// TwinCAT 3 PLC project Controller
// ProgramVersion: 3.1.4020.2
// libraries:
//   Tc2_Standard, * (Beckhoff Automation GmbH)
//   Tc2_System, * (Beckhoff Automation GmbH)
//   Tc2_TcpIp, * (Beckhoff Automation GmbH)
//   Tc2_Utilities, * (Beckhoff Automation GmbH)
//   Tc3_Module, * (Beckhoff Automation GmbH)
// project tree:
//   / GlobalTextList.TcGTLO, ImagePool.TcIPO (not stored), PlcTask.TcTTO, Visualization Manager.TcVMO (not stored), VISU_TASK.TcTTO
//   GVLs/ GVL.TcGVL
//   POUs/Helpers/ FB_FrameFifo.TcPOU, FB_LogFifo.TcPOU
//   POUs/ MAIN.TcPOU
//   POUs/SocketClient/ FB_ProcessSocketData.TcPOU, FB_SocketClient.TcPOU, FB_SocketClientConnection.TcPOU
//   VISUs/ Visualization.TcVIS
// real-time tasks:
//   TASK PlcTask: cycle T#10ms, priority 20, ADS port 350
//   TASK IOTask: cycle T#10ms, priority 1, ADS port 351
//   TASK VISU_TASK: cycle T#200000us, priority 30, ADS port 352

CONFIGURATION Controller
    RESOURCE PLC ON TwinCAT3
        TASK PlcTask(INTERVAL := T#10ms, PRIORITY := 20);
        TASK VISU_TASK(INTERVAL := T#200000us, PRIORITY := 30);
        PROGRAM MAIN WITH PlcTask : MAIN;
        PROGRAM VisuElems_Visu_Prg WITH VISU_TASK : VisuElems.Visu_Prg;
    END_RESOURCE
END_CONFIGURATION

// ---- GVLs/GVL.TcGVL
{attribute 'qualified_only'}
VAR_GLOBAL CONSTANT
	PLCPRJ_BUFFER_SIZE		: UDINT := 1000;					(* Max. internal fifo/receiver buffer size *)
	
	PLCPRJ_CLIENT_SEND_CYCLE_TIME			: TIME := T#1S;
	PLCPRJ_RECEIVE_POLLING_TIME				: TIME := T#100MS;
	PLCPRJ_RECEIVE_TIMEOUT					: TIME := T#50S;
	
	(* Some project specific error codes *)
	PLCPRJ_ERROR_RECEIVE_TIMEOUT			: UDINT := 16#8101;(* Receive timeout *)
	PLCPRJ_ERROR_SENDFIFO_OVERFLOW			: UDINT := 16#8102;(* Send fifo overflow *)
	PLCPRJ_ERROR_RECFIFO_OVERFLOW			: UDINT := 16#8103;(* Receive fifo overflow *)	
	
	TERMINATION_CHAR_CODE					: BYTE := 10;	
	
END_VAR

VAR_GLOBAL
	sSrvNetID					: T_AmsNetID	:= ''; 				(* TwinCAT TCP/IP server network address - Set to Local via ''*)
	sSocketRemoteHost			: T_IPv4Addr := '10.5.1.166';		(* Remote Socket Server IP Address*)
	nSocketRemotePort			: UDINT := 14150;  					(* Server port number *)
	
	RFID_TAG			AT %Q*	: STRING(40);
	READ_ZONE_BEGIN 	AT %I*	: BOOL;
	SET_TEST_OUTPUT		AT %Q* 	: BOOL;
	TON_FLASH					: TON;
	
END_VAR

// ---- POUs/MAIN.TcPOU
PROGRAM MAIN
VAR
	bSocketCloseAll			: BOOL := TRUE;
	fbSocketCloseAll		: FB_SocketCloseAll;
	fbSocketClient			: FB_SocketClient := ( 	sRemoteHost := GVL.sSocketRemoteHost,(* Remote (server) IP address! *)
										nRemotePort := GVL.nSocketRemotePort,(* Remote (server) port number! *)  
										sPrefix := 'CLIENT::' );(* Application (connection) instance *)
										
	bEnableSocket			: BOOL 	:= TRUE;   (* TRUE => enable client data exchange, FALSE => disable *)
	bEnableLogging			: BOOL	:= TRUE;   (* TRUE => Enable message/error log, FALSE => Disable *)
END_VAR

(* On PLC reset or program download close all old (opened) connections *)
fbSocketCloseAll( 	sSrvNetID := GVL.sSrvNetID, 
					bExecute:= bSocketCloseAll );
					
IF fbSocketCloseAll.bBusy OR fbSocketCloseAll.bError THEN
	RETURN;
END_IF
bSocketCloseAll := FALSE;

fbSocketClient( sSrvNetId := GVL.sSrvNetID, 
				bEnable := bEnableSocket, 
				bLog := bEnableLogging );
				
IF GVL.TON_FLASH.Q THEN
	GVL.TON_FLASH( IN := FALSE);
	GVL.SET_TEST_OUTPUT := 0;
END_IF

END_PROGRAM

// ---- POUs/SocketClient/FB_SocketClient.TcPOU
FUNCTION_BLOCK FB_SocketClient
VAR_INPUT
	sSrvNetID	: T_AmsNetID	:= '';(* TwinCAT TCP/IP server network address *)
	sRemoteHost	: T_IPv4Addr 	:= '127.0.0.1';(* Server network address *)
	nRemotePort	: UDINT 		:= 200;(* Server port number *)
	bEnable		: BOOL 			:= FALSE;(* TRUE => enable client data exchange, FALSE => disable *)
	bLog		: BOOL 			:= FALSE;(* TRUE => Enable log message output, FALSE => Disable *)
	sPrefix		: STRING 		:= 'CLIENT::';(* Log message description string (allows the identification of log message source) *)
END_VAR
VAR_OUTPUT
	eState		: E_SocketConnectionState := eSOCKET_DISCONNECTED;(* TCP/IP connection state *)
END_VAR
VAR
	fbProcessSocketData : FB_ProcessSocketData;				(* Client application control function block *)
	fbClientConnection	: FB_SocketClientConnection;		(* Client data exchange control function block *)
	fbTx 				: FB_FrameFifo;						(* Tx fifo *)
	fbRx 				: FB_FrameFifo;						(* Rx fifo *)
	fbLog				: FB_LogFifo;						(* Log/debug/error fifo *)
END_VAR

(*-------------------------- Trigger data exchange -----------------------------------------------*)
fbClientConnection( sSrvNetID := sSrvNetID, fbRx := fbRx, fbTx := fbTx, fbLog := fbLog, 
					bEnable := bEnable, sRemoteHost := sRemoteHost, nRemotePort := nRemotePort,  
					bLog := bLog, sPrefix := sPrefix, eState=>eState );
	
IF fbClientConnection.eState = eSOCKET_CONNECTED THEN (* Connection established *)
	fbProcessSocketData( fbTx := fbTx, fbRx := fbRx, fbLog := fbLog );
END_IF

END_FUNCTION_BLOCK

// ---- POUs/SocketClient/FB_ProcessSocketData.TcPOU
FUNCTION_BLOCK FB_ProcessSocketData
VAR_IN_OUT
	fbTx 		: FB_FrameFifo;(* TX fifo *)
	fbRx 		: FB_FrameFifo;(* RX fifo *)
	fbLog		: FB_LogFifo;(* Log message fifo *)
END_VAR
VAR
	sToServer	: T_MaxString := '';
	sFromServer	: T_MaxString := '';
	sLogMessage : T_MaxString := '';
	nCounter	: UDINT;
	fbSndTimer	: TON;
END_VAR

(*------------------------------- Send cyclic message strings ------------------------------------------*)
fbSndTimer( IN := FALSE, PT := GVL.PLCPRJ_CLIENT_SEND_CYCLE_TIME );
IF fbSndTimer.Q THEN
	fbSndTimer( IN := FALSE );

	(* Create new message string *)
	nCounter := nCounter  + 1;
	sToServer := CONCAT( 'Client message: ', UDINT_TO_STRING(nCounter) );

	fbTx.AddToTail( sPut := sToServer );(* Put string to the tx fifo *)
	IF NOT fbTx.bOk THEN(* TX fifo overflow => log error *)
		fbLog.Error( sMessage := 'FB_FrameFifo(sender)', nErrID := GVL.PLCPRJ_ERROR_SENDFIFO_OVERFLOW );
	END_IF

END_IF

(*------------------------------- Get received message strings ------------------------------------------*)
REPEAT
	fbRx.RemoveFromHead();(* Fetch string from rx fifo *)
	IF fbRx.bOk THEN(* Success *)

		(* TODO: Implement receive data handler *)
		sFromServer := fbRx.sGet;
		
		(* TEST HANDLER *)
		GVL.RFID_TAG := sFromServer;
		IF LEN(sFromServer) > 0 THEN
			GVL.TON_FLASH( IN := TRUE, PT := T#0.25S );		
			GVL.SET_TEST_OUTPUT := 1;	
		END_IF
		sFromServer := '';
		(* END TEST HANDLER *)
		
	END_IF
	
UNTIL NOT fbRx.bOk

END_REPEAT


(*------------------------------- Get log/error messages from log fifo ------------------------------------------*)
REPEAT
	fbLog.Remove( );
	IF fbLog.bOk THEN

		(* TODO: Implement log message handler *)
		sLogMessage := fbLog.sGet;

	END_IF
UNTIL NOT fbLog.bOk
END_REPEAT

END_FUNCTION_BLOCK

// ---- POUs/Helpers/FB_FrameFifo.TcPOU
(* Tx/Rx (string data) fifo control function block *)
FUNCTION_BLOCK FB_FrameFifo
VAR_INPUT
	bLog		: BOOL			:= FALSE;			(* TRUE => Enable log message output, FALSE => Disable *)
	sPrefix		: STRING		:= 'Unknown::';		(* Log message description string (allows the identification of log message source) *)
	sPut		: T_MaxString 	:= ''; 				(* String message to add (write) to the fifo *)
END_VAR
VAR_OUTPUT
	bOk			: BOOL; 	 						(* TRUE = New entry added or removed succesfully, FALSE = Fifo overflow or fifo empty *)
	sGet		: T_MaxString 	:= '';				(* String message removed (read) from fifo *)
	nCount		: UDINT			:= 0;				(* Number of fifo entries *)
	cbFree		: UDINT 		:= 0;				(* Free buffer space *)	
END_VAR
VAR
	fbBuffer 	: FB_StringRingBuffer := (bOverwrite := FALSE);(* Basic (lower level) string buffer control function block *)
	buffer		: ARRAY[-3..GVL.PLCPRJ_BUFFER_SIZE] OF BYTE;(* Internal buffer memory *)	
END_VAR

;

ACTION AddToTail:
(* Adds new fifo entry *)
fbBuffer.A_AddTail( pBuffer:= ADR(buffer), cbBuffer:= SIZEOF(buffer),
					putValue:= sPut, bOk=>bOk, nCount=>nCount );
IF bOk THEN
	cbFree := GVL.PLCPRJ_BUFFER_SIZE - fbBuffer.cbSize;(* Calculate the free buffer space *)
	IF bLog THEN(* Log message *)
		ADSLOGSTR( ADSLOG_MSGTYPE_HINT OR ADSLOG_MSGTYPE_LOG, CONCAT( sPrefix, '<="%s"' ), sPut );
	END_IF
END_IF
END_ACTION

ACTION Clear:
(* Resets fifo = clears all data *)
fbBuffer.A_Reset( pBuffer:= ADR(buffer), cbBuffer:= SIZEOF(buffer),
				bOk=>bOk, getValue=>sGet, nCount=>nCount );
				
cbFree := GVL.PLCPRJ_BUFFER_SIZE;(* Free buffer size *)
END_ACTION

ACTION RemoveFromHead:
(* Removes oldest fifo entry *)
fbBuffer.A_RemoveHead( pBuffer:= ADR(buffer), cbBuffer:= SIZEOF(buffer),
						bOk=>bOk, getValue=>sGet, nCount=>nCount );
IF bOk THEN
	cbFree := GVL.PLCPRJ_BUFFER_SIZE - fbBuffer.cbSize;(* Calculate the free buffer space *)
END_IF
END_ACTION

END_FUNCTION_BLOCK

// ---- POUs/Helpers/FB_LogFifo.TcPOU
(* Log/debug/error message fifo *)
FUNCTION_BLOCK FB_LogFifo
VAR_INPUT
	bLog		: BOOL 		:= FALSE;				(* TRUE => Enable log message output, FALSE => Disable *)
	sPrefix		: STRING 	:= 'Unknown::';			(* Log message description string (allows the identification of log message source) *)
	
	sMessage	: STRING 	:= '';					(* String message to add (write) to the fifo *)
	nErrID		: UDINT 	:= 0;					(* Error code to add (write) to the fifo *)
	hSocket		: T_HSOCKET;						(* Socket connection handle *)
END_VAR
VAR_OUTPUT
	bOk			: BOOL;								(* TRUE = New entry added or removed succesfully, FALSE = Fifo overflow or fifo empty *)
	sGet		: T_MaxString := '';				(* String entry removed (read) from fifo *)
	nCount		: UDINT := 0;						(* Number of fifo entries *)	
END_VAR
VAR
	fbBuffer 	: FB_StringRingBuffer;(* Basic (lower level) string buffer control function block *)
	buffer		: ARRAY[0..GVL.PLCPRJ_BUFFER_SIZE] OF BYTE;(* Internal buffer memory *)
	sSource		: T_MaxString;	
	sPut		: T_MaxString;	
END_VAR

;

ACTION Clear:
(* Clears all fifo entries *)
fbBuffer.A_Reset( 	pBuffer := ADR( buffer ), cbBuffer := SIZEOF( buffer ), 
					bOk=>bOk, nCount=>nCount, getValue=>sGet );
END_ACTION

ACTION Error:
(* Adds new fifo entry *)
IF nErrID = 0 THEN
	sSource := '::Error: 0x';
ELSIF ( nErrID AND 16#80000000) = 16#80000000 THEN
	IF nErrID = 16#80072746 THEN
		sSource := '::Win32 error (the connection is reset by remote side): 0x';
	ELSE
		sSource := '::Win32 error: 0x';
	END_IF
ELSIF (nErrID AND 16#00008100) = 16#00008100 THEN
	CASE nErrID OF
		GVL.PLCPRJ_ERROR_RECEIVE_TIMEOUT:
			sSource := '::PLC sample project receive timeout error: 0x';
		GVL.PLCPRJ_ERROR_SENDFIFO_OVERFLOW:
			sSource := '::PLC sample project send fifo overflow error: 0x';
		GVL.PLCPRJ_ERROR_RECFIFO_OVERFLOW:
			sSource := '::PLC sample project receive fifo overflow error: 0x';
	ELSE
		sSource := '::Other PLC sample project error: 0x';
	END_CASE
ELSIF (nErrID AND 16#00008000) = 16#00008000 THEN
	sSource := '::Internal TCP/IP Connection Server error: 0x';
ELSE
	sSource := '::TwinCAT System error: 0x';
END_IF

sPut := CONCAT( CONCAT( CONCAT( sPrefix, sMessage ), sSource ), DWORD_TO_HEXSTR( nErrID AND 16#FFFF, 0, FALSE ) ); 

fbBuffer.A_AddTail( pBuffer:= ADR(buffer), cbBuffer:= SIZEOF(buffer),
					putValue:= sPut, bOk=>bOk, nCount=>nCount );
IF bOk THEN
	IF bLog THEN(* Log error message *)
		ADSLOGSTR( ADSLOG_MSGTYPE_ERROR OR ADSLOG_MSGTYPE_LOG, '%s', sPut );	
	END_IF
END_IF
END_ACTION

ACTION Message:
(* Adds new fifo entry *)
sPut := CONCAT( CONCAT( sPrefix, sMessage ), CONCAT( '::', HSOCKET_TO_STRING(hSocket) ) );
fbBuffer.A_AddTail( pBuffer:= ADR(buffer), cbBuffer:= SIZEOF(buffer),
					putValue:= sPut, bOk=>bOk, nCount=>nCount );
IF bOk THEN
	IF bLog THEN(* Log information message *)
		ADSLOGSTR( ADSLOG_MSGTYPE_HINT OR ADSLOG_MSGTYPE_LOG, '%s', sPut );	
	END_IF
END_IF
END_ACTION

ACTION Remove:
(* Removes oldest fifo entry *)
IF nCount = 0 THEN
	sGet := '';
	bOk := FALSE;
	RETURN;
END_IF

fbBuffer.A_RemoveHead( pBuffer:= ADR(buffer), cbBuffer:= SIZEOF(buffer),
						getValue=>sGet, bOk=>bOk, nCount=>nCount );
END_ACTION

END_FUNCTION_BLOCK

// ---- POUs/SocketClient/FB_SocketClientConnection.TcPOU
(* This function block implements simple TCP/IP client protocol. *)
FUNCTION_BLOCK FB_SocketClientConnection
VAR_IN_OUT
	fbTx 		: FB_FrameFifo;  (* TX fifo *)
	fbRx 		: FB_FrameFifo;  (* RX fifo *)
	fbLog		: FB_LogFifo;    (* Log message fifo *)
END_VAR

VAR_INPUT
	sSrvNetID	: T_AmsNetID	:= '';				(* TwinCAT TCP/IP server network address *)
	sRemoteHost	: T_IPv4Addr	:= '127.0.0.1';		(* Server network address *)
	nRemotePort	: UDINT			:= 200;				(* Remote server port *)
	bEnable		: BOOL			:= FALSE;			(* TRUE => Enable/connect, FALSE => Disable/disconnect *)
	tReconnect	: TIME 			:= T#10S;			(* Try to reconnect after this time *)
	bLog		: BOOL 			:= FALSE;			(* TRUE => Enable log message output, FALSE => Disable *)
	sPrefix		: STRING 		:= 'CLIENT::';		(* Log message description string (allows the identification of log message source) *)
END_VAR

VAR_OUTPUT
	eState		: E_SocketConnectionState := eSOCKET_DISCONNECTED;		(* TCP/IP connection state *)
END_VAR
VAR
	fbSocketConnect 	: FB_ClientServerConnection;					(* Create/release TCP/IP connection *)
	fbSocketSend		: FB_SocketSend;								(* Send TCP/IP data *)
	fbSocketReceive		: FB_SocketReceive;								(* Receive TCP/IP data *)
	
	nState 		: BYTE;													(* Global state *)
	bSndBusy 	: BOOL;													(* Tx state *)
	bRcvBusy 	: BOOL;													(* Rx state *)
	bDisconnect	: BOOL;													(* Disconnect flag, if set the socket will be closed *)

	fbReceivePollTimer	: TON;											(* Receive poll timer *)
	fbResponseTimer		: TON;											(* Response timeout timer *)
	fbReconnectTimer 	: TON;											(* Reconnect timer *)

	dBytesReceived		: UDINT;										(* Count of received data bytes *)
	dRxLength			: UDINT;										(* Byte length of received string *)
	buffer				: ARRAY[0..GVL.PLCPRJ_BUFFER_SIZE] OF BYTE;		(* Temp. RX buffer *)
	sRxFrame			: T_MaxString;
	sTxFrame			: T_MaxString;
	i					: UDINT;
	bAbort				: BOOL;
END_VAR

CASE nState OF
	0:(* Connect *)
		fbSocketConnect( sSrvNetID 		:= sSrvNetID,
						nMode			:= SEL( bLog, 0, CONNECT_MODE_ENABLEDBG),(* Enable/disable debug messages? *)
						sRemoteHost 	:= sRemoteHost, nRemotePort := nRemotePort,
						bEnable			:= bEnable, tReconnect	:= tReconnect,
						eState			=> eState );
						
		IF NOT fbSocketConnect.bBusy THEN
			IF NOT fbSocketConnect.bError THEN
				IF eState = eSOCKET_CONNECTED THEN   (* We are connected *)
					
					fbTx.Clear( sPrefix := CONCAT( sPrefix, 'FB_FrameFifo(sender)::' ), bLog := bLog );(* Clear TX fifo (optional) *)
					fbRx.Clear( sPrefix := CONCAT( sPrefix, 'FB_FrameFifo(receiver)::' ), bLog := bLog );(* Clear RX fifo (optional) *)
					fbLog.Clear( sPrefix := sPrefix, bLog := bLog );(* Clear log fifo (optional) *)
					bSndBusy := FALSE;
					bRcvBusy := FALSE;
					bDisconnect := FALSE;
					dBytesReceived 	:= 0;

					fbReceivePollTimer( IN := FALSE, PT := T#0S );
					fbResponseTimer( IN := FALSE, PT := GVL.PLCPRJ_RECEIVE_TIMEOUT );
					fbReconnectTimer( IN := FALSE, PT := tReconnect );
				
					fbLog.Message( sMessage := 'Connection established!', hSocket := fbSocketConnect.hSocket );
					nState := 1;
				END_IF
			ELSE(* Connect error => log error *)
				fbLog.Error( sMessage := 'FB_ClientServerConnection()', nErrID := fbSocketConnect.nErrId );
			END_IF
		END_IF


	1:(* Data exchange state *)
		bDisconnect := NOT bEnable OR bDisconnect;(* User/internal disconnect requested? *)
		IF bDisconnect AND NOT bSndBusy AND NOT bRcvBusy THEN
			bDisconnect := FALSE;
			fbLog.Message( sMessage := 'Closing connection!', hSocket := fbSocketConnect.hSocket );
			nState := 2;(* Disconnect *)
		ELSE

			(* ------------------ Send tx data -------------------------------------- *)
			
			IF NOT bDisconnect AND NOT bSndBusy THEN
				fbTx.RemoveFromHead( sGet => sTxFrame );(* Remove oldest string entry *)
				IF fbTx.bOk THEN(* Success *)
					fbSocketSend( bExecute := FALSE );
					fbSocketSend(sSrvNetID 	:= sSrvNetID,
							hSocket		:= fbSocketConnect.hSocket,
							cbLen		:= INT_TO_UDINT(LEN( sTxFrame )) + 1,(* Send string inclusive string (null) delimiter! *)
							pSrc		:= ADR( sTxFrame ),(* Address of the string variable *)
							bExecute	:= TRUE );
					bSndBusy := TRUE;
				END_IF
			ELSE(* Wait until send not busy *)
				fbSocketSend( bExecute := FALSE );
				IF NOT fbSocketSend.bBusy THEN
					bSndBusy := FALSE;
					IF fbSocketSend.bError THEN(* Send error => log error and disconnect *)
						fbLog.Error( sMessage := 'FB_SocketSend()', nErrID := fbSocketSend.nErrId );
						bDisconnect := TRUE;(* Set flag *)
					END_IF
				END_IF
			END_IF  
			(* ---------------------------------------------------------------------- *)


			(* ---------------------- Get rx data ----------------------------------- *)
			IF NOT bDisconnect AND NOT bRcvBusy THEN
				
				fbReceivePollTimer( IN := TRUE );
				IF fbReceivePollTimer.Q THEN
					IF fbRx.cbFree >= SIZEOF(sRxFrame) THEN(* Check free rx fifo space *)
						fbReceivePollTimer( IN := FALSE, PT := GVL.PLCPRJ_RECEIVE_POLLING_TIME );
						fbSocketReceive( bExecute := FALSE );
						fbSocketReceive(sSrvNetId	:= sSrvNetID,
										hSocket		:= fbSocketConnect.hSocket,
										cbLen		:= SIZEOF(buffer) - dBytesReceived,
										pDest		:= ADR(buffer) + dBytesReceived,
										bExecute	:= TRUE );
						bRcvBusy := TRUE;
					END_IF
				END_IF
				
			ELSE(* Wait until receive not busy *)

				fbSocketReceive( bExecute := FALSE );
				IF NOT fbSocketReceive.bBusy THEN
					bRcvBusy := FALSE;
					IF NOT fbSocketReceive.bError THEN
						IF fbSocketReceive.nRecBytes > 0 THEN(* Bytes received *)
							
							fbReceivePollTimer( IN := FALSE, PT := T#0S );(* Bytes received => increase the read (polling) speed *)
							fbResponseTimer( IN := FALSE );(* Bytes received => disable timeout check *)
							dBytesReceived := dBytesReceived + fbSocketReceive.nRecBytes;(* Calculate the number of received data bytes *)

							(* Parse received bytes and extract strings *)
							REPEAT
								bAbort := TRUE;(* set flag *)
								IF dBytesReceived > 0 THEN

									(* Search for string null delimiter *)
									FOR i:= 0 TO dBytesReceived - 1 BY 1 DO
										IF buffer[i] = GVL.TERMINATION_CHAR_CODE THEN (* End of string position found *)

											dRxLength := i + 1;(* Calculate the length of string (inclusive the end delimiter) *)
											MEMCPY( ADR(sRxFrame), ADR(buffer), MIN(dRxLength, SIZEOF(sRxFrame) ) );(* Copy string bytes to temp string variable *)

											fbRx.AddToTail( sPut := sRxFrame );(* Add string to the rx fifo *)
											IF fbRx.bOk THEN
												MEMMOVE( ADR(buffer), ADR(buffer) + dRxLength, dBytesReceived - dRxLength );(* Move/shift remaining bytes in buffer *)
												dBytesReceived := dBytesReceived - dRxLength;(* Recalculate the remaining data length *)

												IF fbRx.cbFree >= SIZEOF(sRxFrame) THEN (* Check free rx buffer space *)
													bAbort := FALSE;(* Reset flag, try to parse the next string *)
												END_IF
											ELSE(* Fifo overflow => log error and disconnect *)
												fbLog.Error( sMessage := 'FB_FrameFifo(receiver)', nErrID := GVL.PLCPRJ_ERROR_RECFIFO_OVERFLOW );
												bDisconnect := TRUE;(* set flag *)
												RETURN;
											END_IF

											EXIT;
										END_IF
									END_FOR

								END_IF (* IF cbReceived > 0 THEN *)

							UNTIL bAbort
							END_REPEAT

						ELSE(* No bytes received *)
							fbResponseTimer( IN := TRUE );(* No bytes received => enable timeout check *)
							IF fbResponseTimer.Q THEN (* Timeout error*)
								fbResponseTimer( IN := FALSE );
								fbLog.Error( sMessage := 'FB_SocketReceive()', nErrID := GVL.PLCPRJ_ERROR_RECEIVE_TIMEOUT );
								bDisconnect := TRUE;(* Set flag *)
							END_IF							
						END_IF(* IF fbReceive.nRecBytes > 0 THEN *)
					ELSE(* Receive error => log error and disconnect *)
						fbLog.Error( sMessage := 'FB_SocketReceive()', nErrID := fbSocketReceive.nErrId );
						bDisconnect := TRUE;(* set flag *)
					END_IF
					
				END_IF(* IF NOT fbReceive.bBusy THEN *) 
	
			END_IF(* IF NOT bDisconnect AND NOT bRcvBusy THEN *)
			(* ---------------------------------------------------------------------- *)
			

		END_IF(* IF bDisconnect AND NOT bSndBusy AND NOT bRcvBusy THEN *)


	2:(* Disconnect *)
		fbSocketConnect( bEnable:= FALSE, eState=>eState );
		IF eState = eSOCKET_DISCONNECTED THEN
			fbReconnectTimer( IN := TRUE );(* Please wait some seconds and then try to connect again *)
			IF fbReconnectTimer.Q THEN
				fbReconnectTimer( IN := FALSE );
				nState := 0;
			END_IF
		END_IF

END_CASE

END_FUNCTION_BLOCK

// ---- GlobalTextList.TcGTLO
TEXTLIST GlobalTextList
  0 = '%s'
END_TEXTLIST

// ---- VISUs/Visualization.TcVIS
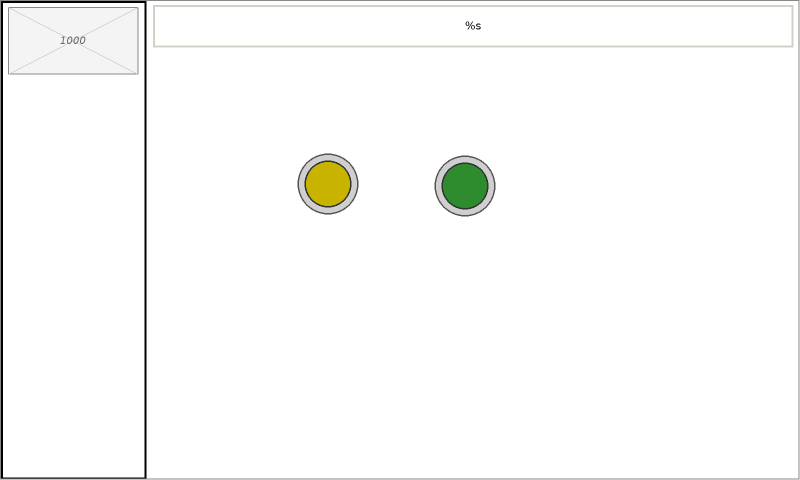
VISUALIZATION Visualization  // 800x480
    Rectangle (1,1 145x478)
    Lamp1 (430,151 70x70), variable: GVL.SET_TEST_OUTPUT, style: Lamp-Lamp1-Green
    Lamp1 (293,149 70x70), variable: GVL.SET_TEST_OUTPUT, style: Lamp-Lamp1-Yellow
    Textfield (153,5 640x42), "%s", text variable: GVL.RFID_TAG
    Image (8,7 130x67), image: 1000
END_VISUALIZATION
